# EPICS substitutions: exampleTop/DeviceDbApp/UaDemoServerDb/UaDemoServer-server.substitutions
file opcuaServerInfo.template {
{ P=$(P=), R=$(R=), SESS=$(SESS) }
}

file opcuaServerStats.template {
{ P=$(P=), R=$(R=), SESS=$(SESS), SUBS=$(SUBS) }
}
